TYPE ST_CtrlInMovableStop :
STRUCT
	ExternalTrigger			: BOOL;
	
END_STRUCT
END_TYPE

(* stored: Version 1.1.0.1, ProductVersion 3.1.4024.9
   DUT ST_CtrlInMovableStop: Id {694c60dd-e96f-4bbd-8c56-32ecfdfad9e8} *)
